{attribute 'GeneratedUsingTerminal: EL6688-0000-0016'}
{attribute addProperty BoxType "EL6688-0000-0016"}
{attribute addProperty Id "Sync_ModeAT %I*BYTE1Control_value_update_toggleAT %I*BOOL1Time_stamp_update_toggleAT %I*BOOL1External_device_not_connectedAT %I*BOOL1"}
{attribute addProperty CRC "2534691805"}
{attribute addProperty Size "4"}
TYPE SYNC_Inputs_971453DD :
STRUCT
	{attribute addProperty Name "Sync_Mode"}
	Sync_Mode AT %I* : BYTE;
	{attribute addProperty Name "Control_value_update_toggle"}
	Control_value_update_toggle AT %I* : BOOL;
	{attribute addProperty Name "Time_stamp_update_toggle"}
	Time_stamp_update_toggle AT %I* : BOOL;
	{attribute addProperty Name "External_device_not_connected"}
	External_device_not_connected AT %I* : BOOL;
END_STRUCT
END_TYPE

(* stored: Version 1.2.0.0, ProductVersion 3.1.4024.9
   DUT SYNC_Inputs_971453DD: Id {352f3687-d545-4eb7-a0bf-88f94fe01aa3} *)
